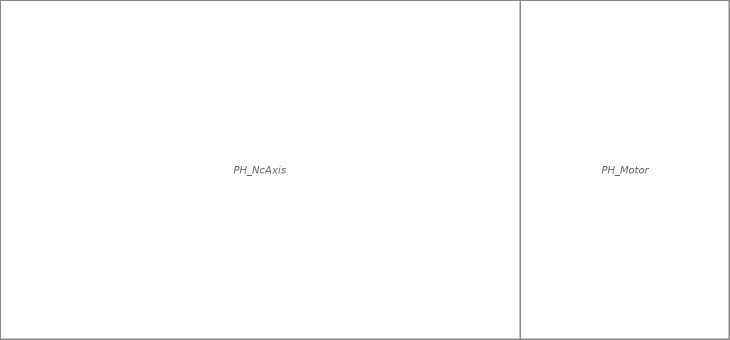
VISUALIZATION PH_AxisOnline  // 730x340
//==================================================================================================
//							Beckhoff Automation Poland
//									18.04.2018
//	Wizualizacja dla Axis Online
//  v1.0	|| TC v 3.1.4022.16		|| - pierwsza wersja
//==================================================================================================
VAR_IN_OUT
	stMcAxisOnline			: ST_McAxisOnline;	
END_VAR
    Frame (0,0 520x340)
        shows PH_NcAxis(stMcAxisOnline := stMcAxisOnline)
    Frame (520,0 210x340)
        shows PH_Motor(stMcAxisOnline := stMcAxisOnline)
END_VISUALIZATION

(* stored: Version 1.1.0.1, ProductVersion 3.1.4022.10
   Visu PH_AxisOnline: Id {0410f5e5-a7d7-4e6b-9a19-4056a2bb405e} *)
